VAR_GLOBAL CONSTANT
	MAX_STRING_LENGTH: INT := 255;
ENd_VAR

(* stored: Version 1.1.0.1, ProductVersion 3.1.4024.9
   GVL GENERAL: Id {dd3625dd-e2db-4fe9-bc13-d46ea5bb5514} *)
